_CFC_ (* Continuous Function Chart, elements in execution order *)
#0 FT_Ostanov:F_TRIG(CLK: SCHU_P2_1_UST_RE_OSTANOV)
#1 TOF_Progrev:TOF(IN: SCHU_P2_1_UST_RE_PROGREV, PT: T#1s)
#2 AND(#1.Q, SCHU_P2_1_UST_SOST_OTKL)
#3 AND(M1_OTKAZ, M2_OTKAZ)
#4 OR(NOT SCHU_P2_1_K1_DI6_FIRE, SCHU_P2_1_Z_NET_VH_NAPR, #0.Q, SCHU_P2_1_Z_GVS1_OTKAZ, #2, SCHU_P2_1_HZ20S60, Z_ZAM_SR, #3, #3, SCHU_P2_1_Z_YA1_OTKAZ, SCHU_P2_1_Z_OTKAZ_VTORICH_SEP, SCHU_P2_1_Z_PREVDAV, SCHU_P2_1_Z_NetP)
#5 SCHU_P2_1_UST_SET_STOP <= #4
#6 sr_stop:SR(SET1: #4, RESET: SCHU_P2_1_UST_SOST_VKL)
#7 SCHU_P2_1_UST_RE_STOP <= #6.Q1
_END_CFC_
(* the same logic as Structured Text *)
FT_Ostanov(CLK := SCHU_P2_1_UST_RE_OSTANOV);
TOF_Progrev(IN := SCHU_P2_1_UST_RE_PROGREV, PT := T#1s);
_t19 := NOT SCHU_P2_1_K1_DI6_FIRE OR SCHU_P2_1_Z_NET_VH_NAPR OR FT_Ostanov.Q OR SCHU_P2_1_Z_GVS1_OTKAZ OR (TOF_Progrev.Q AND SCHU_P2_1_UST_SOST_OTKL) OR SCHU_P2_1_HZ20S60 OR Z_ZAM_SR OR (M1_OTKAZ AND M2_OTKAZ) OR (M1_OTKAZ AND M2_OTKAZ) OR SCHU_P2_1_Z_YA1_OTKAZ OR SCHU_P2_1_Z_OTKAZ_VTORICH_SEP OR SCHU_P2_1_Z_PREVDAV OR SCHU_P2_1_Z_NetP;
SCHU_P2_1_UST_SET_STOP := _t19;
sr_stop(SET1 := _t19, RESET := SCHU_P2_1_UST_SOST_VKL);
SCHU_P2_1_UST_RE_STOP := sr_stop.Q1;
END_PROGRAM

(* POU Regim/Ostanov, CFC *)
PROGRAM Ostanov
VAR
	RT_OTKL: R_TRIG;
	SR_OSTANOV: SR;
	TON_AVR_M: TON;
	Z_zam_ostatov: R_TRIG;
END_VAR
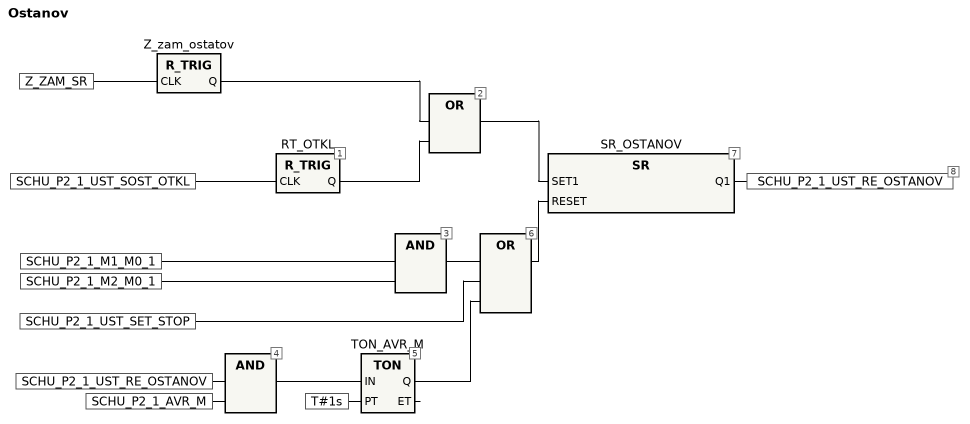
_CFC_ (* Continuous Function Chart, elements in execution order *)
#0 Z_zam_ostatov:R_TRIG(CLK: Z_ZAM_SR)
#1 RT_OTKL:R_TRIG(CLK: SCHU_P2_1_UST_SOST_OTKL)
#2 OR(#0.Q, #1.Q)
#3 AND(SCHU_P2_1_M1_M0_1, SCHU_P2_1_M2_M0_1)
#4 AND(SCHU_P2_1_UST_RE_OSTANOV, SCHU_P2_1_AVR_M)
#5 TON_AVR_M:TON(IN: #4, PT: T#1s)
#6 OR(#3, SCHU_P2_1_UST_SET_STOP, #5.Q)
#7 SR_OSTANOV:SR(SET1: #2, RESET: #6)
#8 SCHU_P2_1_UST_RE_OSTANOV <= #7.Q1
_END_CFC_
(* the same logic as Structured Text *)
Z_zam_ostatov(CLK := Z_ZAM_SR);
RT_OTKL(CLK := SCHU_P2_1_UST_SOST_OTKL);
TON_AVR_M(IN := SCHU_P2_1_UST_RE_OSTANOV AND SCHU_P2_1_AVR_M, PT := T#1s);
SR_OSTANOV(SET1 := Z_zam_ostatov.Q OR RT_OTKL.Q, RESET := (SCHU_P2_1_M1_M0_1 AND SCHU_P2_1_M2_M0_1) OR SCHU_P2_1_UST_SET_STOP OR TON_AVR_M.Q);
SCHU_P2_1_UST_RE_OSTANOV := SR_OSTANOV.Q1;
END_PROGRAM

(* POU Regim/Progrev, CFC *)
PROGRAM Progrev
VAR
	RS_Progrev: RS;
	RT_VKL: R_TRIG;
	TON_SCHU_P2_1_TE2_M_UST: TON;
	SR_First_On: SR;
END_VAR
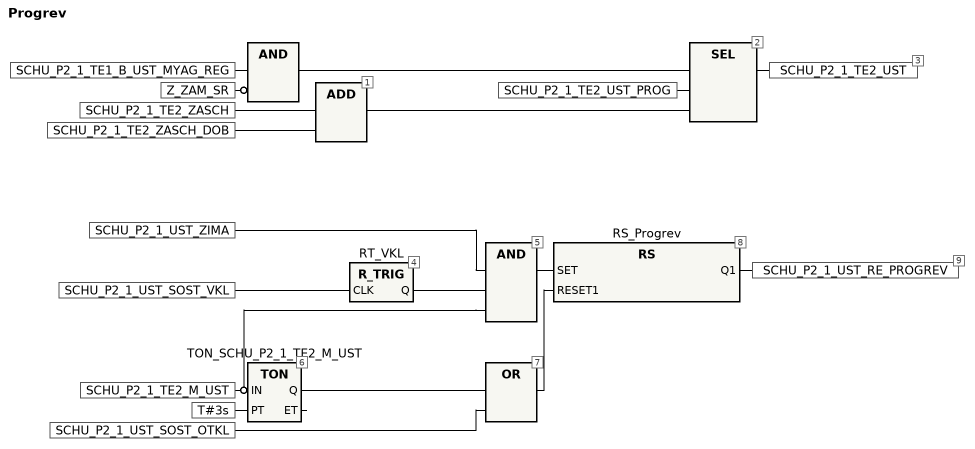
_CFC_ (* Continuous Function Chart, elements in execution order *)
#0 AND(SCHU_P2_1_TE1_B_UST_MYAG_REG, NOT Z_ZAM_SR)
#1 ADD(SCHU_P2_1_TE2_ZASCH, SCHU_P2_1_TE2_ZASCH_DOB)
#2 SEL(#0, SCHU_P2_1_TE2_UST_PROG, #1)
#3 SCHU_P2_1_TE2_UST <= #2
#4 RT_VKL:R_TRIG(CLK: SCHU_P2_1_UST_SOST_VKL)
#5 AND(SCHU_P2_1_UST_ZIMA, #4.Q, SCHU_P2_1_TE2_M_UST)
#6 TON_SCHU_P2_1_TE2_M_UST:TON(IN: NOT SCHU_P2_1_TE2_M_UST, PT: T#3s)
#7 OR(#6.Q, SCHU_P2_1_UST_SOST_OTKL)
#8 RS_Progrev:RS(SET: #5, RESET1: #7)
#9 SCHU_P2_1_UST_RE_PROGREV <= #8.Q1
_END_CFC_
(* the same logic as Structured Text *)
SCHU_P2_1_TE2_UST := SEL(SCHU_P2_1_TE1_B_UST_MYAG_REG AND NOT Z_ZAM_SR, SCHU_P2_1_TE2_UST_PROG, SCHU_P2_1_TE2_ZASCH + SCHU_P2_1_TE2_ZASCH_DOB);
RT_VKL(CLK := SCHU_P2_1_UST_SOST_VKL);
TON_SCHU_P2_1_TE2_M_UST(IN := NOT SCHU_P2_1_TE2_M_UST, PT := T#3s);
RS_Progrev(SET := SCHU_P2_1_UST_ZIMA AND RT_VKL.Q AND SCHU_P2_1_TE2_M_UST, RESET1 := TON_SCHU_P2_1_TE2_M_UST.Q OR SCHU_P2_1_UST_SOST_OTKL);
SCHU_P2_1_UST_RE_PROGREV := RS_Progrev.Q1;
END_PROGRAM

(* POU Regim/Pusk, CFC *)
PROGRAM Pusk
VAR
	RS_Pusk: RS;
	FT_PROGREV: F_TRIG;
	RT_VKL: R_TRIG;
	TON_sost_VKL: TON;
	TON_AVR_M: TON;
	re_start: F_TRIG;
	TON_Z_ZAM: TON;
END_VAR
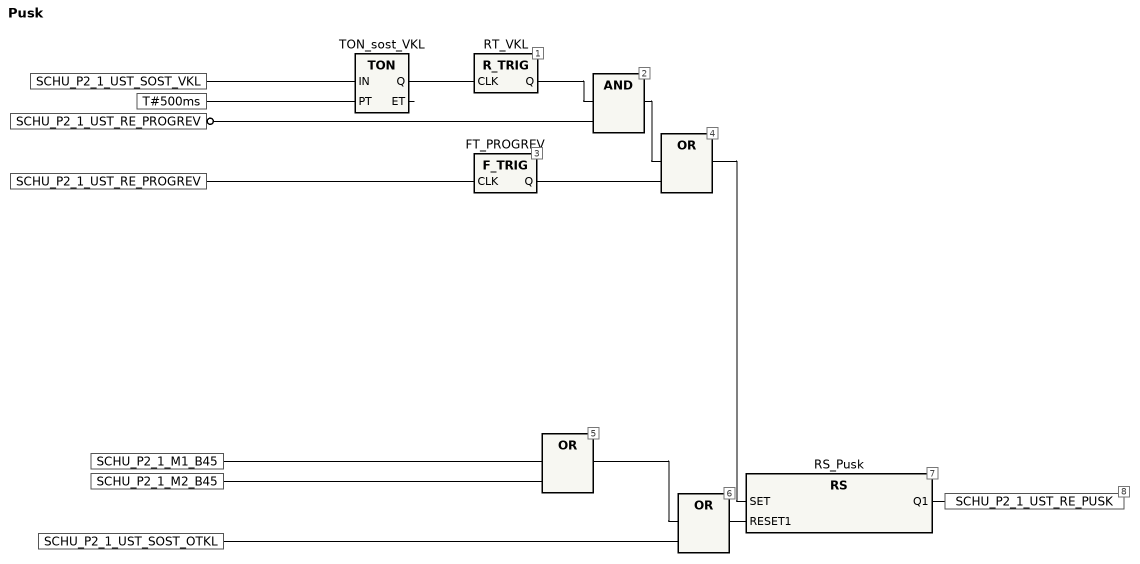
_CFC_ (* Continuous Function Chart, elements in execution order *)
#0 TON_sost_VKL:TON(IN: SCHU_P2_1_UST_SOST_VKL, PT: T#500ms)
#1 RT_VKL:R_TRIG(CLK: #0.Q)
#2 AND(#1.Q, NOT SCHU_P2_1_UST_RE_PROGREV)
#3 FT_PROGREV:F_TRIG(CLK: SCHU_P2_1_UST_RE_PROGREV)
#4 OR(#2, #3.Q)
#5 OR(SCHU_P2_1_M1_B45, SCHU_P2_1_M2_B45)
#6 OR(#5, SCHU_P2_1_UST_SOST_OTKL)
#7 RS_Pusk:RS(SET: #4, RESET1: #6)
#8 SCHU_P2_1_UST_RE_PUSK <= #7.Q1
_END_CFC_
(* the same logic as Structured Text *)
TON_sost_VKL(IN := SCHU_P2_1_UST_SOST_VKL, PT := T#500ms);
RT_VKL(CLK := TON_sost_VKL.Q);
FT_PROGREV(CLK := SCHU_P2_1_UST_RE_PROGREV);
RS_Pusk(SET := (RT_VKL.Q AND NOT SCHU_P2_1_UST_RE_PROGREV) OR FT_PROGREV.Q, RESET1 := (SCHU_P2_1_M1_B45 OR SCHU_P2_1_M2_B45) OR SCHU_P2_1_UST_SOST_OTKL);
SCHU_P2_1_UST_RE_PUSK := RS_Pusk.Q1;
END_PROGRAM

(* POU Regim/Rabota, CFC *)
PROGRAM Rabota
VAR
	RS_Rabota: RS;
	FT_Pusk: F_TRIG;
END_VAR
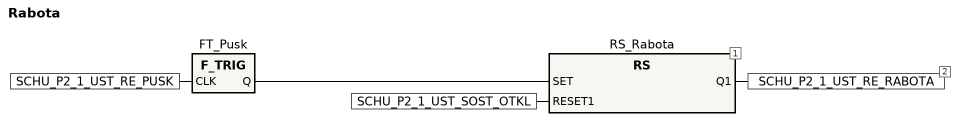
_CFC_ (* Continuous Function Chart, elements in execution order *)
#0 FT_Pusk:F_TRIG(CLK: SCHU_P2_1_UST_RE_PUSK)
#1 RS_Rabota:RS(SET: #0.Q, RESET1: SCHU_P2_1_UST_SOST_OTKL)
#2 SCHU_P2_1_UST_RE_RABOTA <= #1.Q1
_END_CFC_
(* the same logic as Structured Text *)
FT_Pusk(CLK := SCHU_P2_1_UST_RE_PUSK);
RS_Rabota(SET := FT_Pusk.Q, RESET1 := SCHU_P2_1_UST_SOST_OTKL);
SCHU_P2_1_UST_RE_RABOTA := RS_Rabota.Q1;
END_PROGRAM

(* POU IM/ALL_IM, CFC *)
PROGRAM ALL_IM
VAR
END_VAR
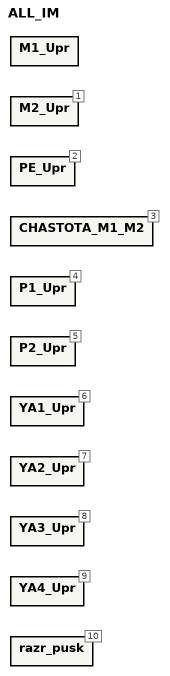
_CFC_ (* Continuous Function Chart, elements in execution order *)
#0 M1_Upr()
#1 M2_Upr()
#2 PE_Upr()
#3 CHASTOTA_M1_M2()
#4 P1_Upr()
#5 P2_Upr()
#6 YA1_Upr()
#7 YA2_Upr()
#8 YA3_Upr()
#9 YA4_Upr()
#10 razr_pusk()
_END_CFC_
(* the same logic as Structured Text *)
M1_Upr();
M2_Upr();
PE_Upr();
CHASTOTA_M1_M2();
P1_Upr();
P2_Upr();
YA1_Upr();
YA2_Upr();
YA3_Upr();
YA4_Upr();
razr_pusk();
END_PROGRAM

(* POU IM/M1_Upr, CFC *)
PROGRAM M1_Upr
VAR
	RS_M1: RS;

	startDelay_M1: TIME := T#0s;
	stopDelay_M1: TIME := T#0s;
	delayFBC_M1: TIME := T#30S;
	feedbPT_M1: TIME := T#120s;
	delayFBP_M1: TIME := T#30s;

	fb_HVACMS_M1: FB_HVACMotor1Speed;
	fb_HVACPIDC_M1: FB_HVACPIDCtrl;

	deadRange: REAL := 0.1;
	rKp: REAL := 1;
	tTi: TIME;
	tTv: TIME := T#0s;
	tTd: TIME := T#0s;
	direction: BOOL;
	rYMin: REAL;
	Dint_Ti: DINT;
	set: BOOL;
	reset: BOOL;
	resetContr: BOOL;
	SR_VKL: SR;
END_VAR
